(* IEC 61131-3 sources: generating_plc_code_with_llms/Code#2/ChatGPT_3.5/first run, 21 files *)

(* ---- 14.st ---- *)
// 8.02s
// 2
FUNCTION FC1001 : BOOL
VAR_INPUT
	MEW: REAL;
	SP: REAL;
	HYS: REAL;
END_VAR

VAR_IN_OUT
	OUT: BOOL;
END_VAR

VAR
	P_HYS: REAL;
END_VAR

(* FC1001 function implementation *)
IF MEW > (SP + P_HYS) THEN
    OUT := TRUE;
ELSIF MEW < (SP - P_HYS) THEN
    OUT := FALSE;
END_IF;

(* Update the hysteresis for the next cycle *)
P_HYS := SP * HYS / 100;

(* Return the output state *)
RETURN OUT;

(* ---- 15.st ---- *)
// 8.78s
// 2
FUNCTION FC1002 : BOOL
VAR_INPUT
	E_A, SENSOR: BOOL;
	ZEITW: TIME;
END_VAR

VAR_IN_OUT
	ZEIT: TON;
	P_HU, P_AL: BOOL;
END_VAR

(* FC1002 function implementation *)
IF E_A THEN
    IF SENSOR THEN
        ZEIT(IN := TRUE, PT := ZEITW);
        P_HU := NOT ZEIT.Q;
        P_AL := ZEIT.Q;
    ELSE
        ZEIT(IN := FALSE);
        P_HU := FALSE;
        P_AL := FALSE;
    END_IF;
ELSE
    ZEIT(IN := FALSE);
    P_HU := FALSE;
    P_AL := FALSE;
END_IF;

(* Return the output state *)
RETURN E_A;

(* ---- 18.st ---- *)
// 7.1s
// 4
FUNCTION FC1003 : VOID
VAR_INPUT
    IN_R: REAL;
    IN_MAX, IN_MIN: REAL;
    OUT_MAX, OUT_MIN: REAL;
END_VAR
VAR_OUTPUT
    OUT_R: REAL;
    FEH: BOOL;
END_VAR
VAR_TEMP
    DIFF1, DIFF2: REAL;
END_VAR

(* Check if input is within the specified range *)
IF (IN_R >= IN_MIN) AND (IN_R <= IN_MAX) THEN
    (* Calculate the differences between the input and output ranges *)
    DIFF1 := OUT_MAX - OUT_MIN;
    DIFF2 := IN_MAX - IN_MIN;

    (* Calculate the scaled temperature value within the output range *)
    OUT_R := OUT_MIN + ((IN_R - IN_MIN) / DIFF2) * DIFF1;

    (* Set FEH (Function Executed Healthy) to TRUE *)
    FEH := TRUE;
ELSE
    (* Set FEH to FALSE if input is outside the specified range *)
    FEH := FALSE;
END_IF

(* ---- 19.st ---- *)
// 10.82s
// 2
FUNCTION_BLOCK FB1005
VAR_INPUT
    START: BOOL;
    DICKE, V_MAX, V_MIN: REAL;
END_VAR

VAR_OUTPUT
    D_MAX, D_MIN: REAL;
    P1: BOOL;
END_VAR

VAR
    FO: BOOL;
    M_MAX, M_MIN: REAL;
END_VAR

METHOD CheckThickness: BOOL
VAR_INPUT
    S1: BOOL;
END_VAR
VAR
    CurrentThickness: REAL;
BEGIN
    (* Check if the sensor is active *)
    IF S1 THEN
        (* Calculate the thickness from the difference of laser measurements *)
        CurrentThickness := DICKE;

        (* Update the maximum and minimum thickness values *)
        IF CurrentThickness > M_MAX THEN
            M_MAX := CurrentThickness;
        END_IF;

        IF CurrentThickness < M_MIN THEN
            M_MIN := CurrentThickness;
        END_IF;

        (* Check if the current thickness is outside the tolerance band *)
        IF CurrentThickness > V_MAX OR CurrentThickness < V_MIN THEN
            P1 := TRUE; (* Switch on the reject light *)
        ELSE
            P1 := FALSE; (* Switch off the reject light *)
        END_IF;
    END_IF;

    (* Output the maximum and minimum thickness values *)
    D_MAX := M_MAX;
    D_MIN := M_MIN;

    (* Reset the thickness values at the start of a new measurement *)
    IF NOT S1 THEN
        M_MAX := 0.0;
        M_MIN := 9999.0; (* Assign an initial large value for comparison *)
    END_IF;

    (* Return the status of the reject light *)
    RETURN P1;
END_METHOD

END_FUNCTION_BLOCK

(* ---- 20.st ---- *)
// 11.08s
// 2
FUNCTION_BLOCK INTERLOCK
    VAR_INPUT
        I1: BOOL;
        I2: BOOL;
        TL: TIME;
    END_VAR

    VAR_OUTPUT
        Q1: BOOL;
        Q2: BOOL;
    END_VAR

    VAR
        T1: TOF(TL);
        T2: TOF(TL);
    END_VAR

    (* Interlock logic *)
    T1(IN:=NOT Q2 AND I1);
    T2(IN:=NOT Q1 AND I2);

    Q1 := T1.Q;
    Q2 := T2.Q;

END_FUNCTION_BLOCK

(* ---- 21.st ---- *)
// 47.97s
// weiter generieren
// 2
FUNCTION_BLOCK BURNER
VAR_INPUT
    IN: BOOL;
    STAGE2: BOOL;
    OVER_TEMP: BOOL;
    OIL_TEMP: BOOL := TRUE;
    FLAME: BOOL;
    RST: BOOL;
    RST_TIMER: BOOL;
    PRE_HEAT_TIME: TIME := t#5s;
    PRE_VENT_TIME: TIME := t#15s;
    PRE_IGNITE_TIME: TIME := t#15s;
    POST_IGNITE_TIME: TIME := t#25s;
    STAGE2_DELAY: TIME := t#10s;
    SAFETY_TIME: TIME := t#5s;
    LOCKOUT_TIME: TIME := t#10s;
    MULTIPLE_IGNITION: BOOL := TRUE;
    KW1: REAL;
    KW2: REAL;
END_VAR
VAR_OUTPUT
    MOTOR: BOOL;
    COIL1: BOOL;
    COIL2: BOOL;
    PRE_HEAT: BOOL;
    IGNITE: BOOL;
    FAIL: BOOL;
    KWH: REAL;
    STATUS: BYTE;
END_VAR
VAR_IN_OUT
    RUNTIME1: UDINT;
    RUNTIME2: UDINT;
    CYCLES: UDINT;
END_VAR
VAR
    state: INT;
    last: TIME;
    tx: TIME;
    last_change: TIME;
    timer1: TON;
    timer2: TON;
    oil_temp_last: BOOL;
    cycles2: UDINT;
END_VAR

METHOD BurnerControl: BOOL
    (* Internal Function to Control Burner *)
    VAR
        t1, t2, t3, t4, t5, t6: TIME;
    END_VAR

    t1 := PRE_HEAT_TIME;
    t2 := t1 + PRE_VENT_TIME;
    t3 := t2 + PRE_IGNITE_TIME;
    t4 := t3 + SAFETY_TIME;
    t5 := t4 + POST_IGNITE_TIME;
    t6 := t5 + STAGE2_DELAY;

    CASE state OF
        110:
            (* Wait for Start Signal (Standby) *)
            IF IN THEN
                state := 111;  (* Move to Startup Sequence *)
                last_change := tx;
            END_IF;
        111:
            (* Startup Sequence *)
            IF NOT OVER_TEMP THEN
                IF (NOT MULTIPLE_IGNITION AND timer1.IN) OR (MULTIPLE_IGNITION) THEN
                    (* Fuel Oil Warming *)
                    PRE_HEAT := TRUE;
                    IF (NOT OIL_TEMP AND (tx - last_change) <= PRE_HEAT_TIME) THEN
                        FAIL := TRUE;  (* Error: Fuel Oil Warming not responded within PRE_HEAT_TIME *)
                        STATUS := 1;
                        RETURN FALSE;
                    END_IF;
                    PRE_HEAT := FALSE;
                ELSE
                    FAIL := TRUE;  (* Error: Flame Sensor active during Fuel Oil Warming *)
                    STATUS := 2;
                    RETURN FALSE;
                END_IF;

                (* Pre-Purge (PRE_VENT_TIME) *)
                MOTOR := TRUE;
                COIL1 := TRUE;
                timer1(IN := TRUE, PT := t2);
                IF (FLAME AND (tx - last_change) <= PRE_VENT_TIME) THEN
                    FAIL := TRUE;  (* Error: Flame Sensor active during Pre-Purge *)
                    STATUS := 3;
                    RETURN FALSE;
                END_IF;

                (* Ignition *)
                COIL1 := FALSE;
                COIL2 := TRUE;
                IGNITE := TRUE;
                timer1(IN := TRUE, PT := t3);
                IF (NOT FLAME AND (tx - last_change) >= SAFETY_TIME) THEN
                    FAIL := TRUE;  (* Error: Safety time passed without flame *)
                    STATUS := 4;
                    RETURN FALSE;
                END_IF;
                IGNITE := FALSE;
                COIL2 := FALSE;
            END_IF;

            (* Stage 1 *)
            IF (tx - last_change) >= t4 THEN
                state := 112;
                last_change := tx;
            END_IF;
        112:
            (* Burner runs at Stage 1 *)
            MOTOR := TRUE;
            COIL1 := TRUE;
            timer1(IN := TRUE);
            KWH := KWH + KW1 * timer1.PT;
            RUNTIME1 := timer1.ET;
            IF (NOT FLAME) THEN
                FAIL := TRUE;  (* Error: Flame stops in operation *)
                STATUS := 5;
                RETURN FALSE;
            END_IF;

            (* Multiple Ignition *)
            IF (FLAME AND MULTIPLE_IGNITION AND (tx - last_change) <= POST_IGNITE_TIME) THEN
                state := 111;  (* Immediately start ignition for stage 1 *)
            END_IF;

            (* Stage 2 Activation *)
            IF STAGE2 AND (tx - last_change) >= t6 THEN
                state := 113;
                last_change := tx;
            END_IF;
        113:
            (* Burner runs at Stage 2 *)
            MOTOR := TRUE;
            COIL2 := TRUE;
            timer2(IN := TRUE);
            KWH := KWH + KW2 * timer2.PT;
            RUNTIME2 := timer2.ET;
    END_CASE;

    (* Check for RST (Reset) *)
    IF RST THEN
        IF (tx - last_change) >= LOCKOUT_TIME AND NOT RST_TIMER THEN
            RST_TIMER := TRUE;  (* Lockout Time Passed, Allow Reset *)
        END_IF;

        IF RST_TIMER THEN
            state := 110;  (* Reset, return to Standby *)
            last_change := tx;
            RST_TIMER := FALSE;
            CYCLES := CYCLES + 1;
        END_IF;
    END_IF;

    (* Check for Over-Temperature *)
    IF OVER_TEMP THEN
        state := 110;  (* Stop immediately every action and report error 9 *)
        FAIL := TRUE;
        STATUS := 9;
    END_IF;

    (* Update STATUS Output *)
    CASE state OF
        110: STATUS := 110;
        111: STATUS := 111;
        112: STATUS := 112;
        113: STATUS := 113;
    END_CASE;

    RETURN TRUE;
END_METHOD;

(* ---- 1.st ---- *)
// 6.53s
// 3
VAR
    xAllOn : BOOL;
    xAllOff : BOOL;

    xAlarm1 : BOOL;
    xAlarm2 : BOOL;
END_VAR

xAllOn := FALSE;
xAllOff := FALSE;
xAlarm1 := FALSE;
xAlarm2 := FALSE;

IF xAllOn THEN
    xAlarm1 := TRUE;
    xAlarm2 := TRUE;
    xAllOn := FALSE;  (* Turn off the xAllOn signal *)
END_IF;

IF xAllOff THEN
    xAlarm1 := FALSE;
    xAlarm2 := FALSE;
    xAllOff := FALSE;  (* Turn off the xAllOff signal *)
END_IF;

(* ---- 10.st ---- *)
// 5.01s
// 4
VAR_INPUT
    X : REAL;
END_VAR

VAR
    result : REAL;
END_VAR

(* Sigmoid function implementation *)
result := 1.0 / (1.0 + EXP(-X));

(* ---- 11.st ---- *)
// 4.88s
// 4
VAR_INPUT
    x : REAL;
END_VAR

VAR
    result : INT;
END_VAR

(* Sign function implementation *)
IF x > 0 THEN
    result := 1;
ELSIF x < 0 THEN
    result := -1;
ELSE
    result := 0;
END_IF;

(* ---- 12.st ---- *)
// 5.26s
// 4
VAR
    X : REAL;
END_VAR

VAR
    result : REAL;
END_VAR

(* Hyperbolic sine function implementation *)
result := (EXP(X) - EXP(-X)) / 2.0;

(* ---- 13.st ---- *)
// 7.85s
// 2
VAR CONSTANT
    MAXNUMBERS : UINT := 99;
END_VAR

VAR
    aNumbers : ARRAY[0..MAXNUMBERS] OF INT;
    nCnt : INT;
END_VAR

VAR
    NumberToFind : INT := 10;
    bNumberFound : BOOL := FALSE;
END_VAR

(* Initialize array with random numbers for illustration purposes *)
FOR nCnt := 0 TO MAXNUMBERS DO
    aNumbers[nCnt] := RAND(1, 20); (* Replace with actual logic for generating random numbers *)
END_FOR;

(* Search for the specific number in the list *)
nCnt := 0;
REPEAT
    IF aNumbers[nCnt] = NumberToFind THEN
        bNumberFound := TRUE;
        EXIT;
    END_IF;
    nCnt := nCnt + 1;
UNTIL nCnt > MAXNUMBERS OR bNumberFound;

(* Check if the number was found or the end of the list is reached *)
IF bNumberFound THEN
    (* Number found *)
    // Your logic here
ELSE
    (* Number not found in the list *)
    // Your logic here
END_IF;

(* ---- 16.st ---- *)
// 12.43s
// 2
VAR
    North_green : BOOL;
    North_yellow : BOOL;
    North_red : BOOL;
    East_green : BOOL;
    East_yellow : BOOL;
    East_red : BOOL;
    T1 : TON;
END_VAR

T1(IN:=TRUE, PT:=10000); (* 10-second cycle *)

IF T1.Q THEN
    (* Between 0ms and 5000ms *)
    IF T1.ET < 5000 THEN
        North_green := TRUE;
        North_yellow := FALSE;
        North_red := FALSE;
        East_green := FALSE;
        East_yellow := FALSE;
        East_red := TRUE;

    (* Between 5000ms and 5500ms *)
    ELSIF T1.ET < 5500 THEN
        North_green := FALSE;
        North_yellow := TRUE;
        North_red := FALSE;
        East_green := FALSE;
        East_yellow := FALSE;
        East_red := TRUE;

    (* Between 5500ms and 9500ms *)
    ELSIF T1.ET < 9500 THEN
        North_green := FALSE;
        North_yellow := FALSE;
        North_red := TRUE;
        East_green := TRUE;
        East_yellow := FALSE;
        East_red := FALSE;

    (* Between 9500ms and 10000ms *)
    ELSE
        North_green := FALSE;
        North_yellow := FALSE;
        North_red := TRUE;
        East_green := FALSE;
        East_yellow := TRUE;
        East_red := FALSE;
    END_IF;
ELSE
    (* Reset lights when the timer is not active *)
    North_green := FALSE;
    North_yellow := FALSE;
    North_red := FALSE;
    East_green := FALSE;
    East_yellow := FALSE;
    East_red := FALSE;
END_IF

(* ---- 17.st ---- *)
// 6.11s
// 4
VAR
    aiOutside : INT;
    aiHumidity: INT;
    sShowText : STRING[80];
END_VAR

(* Weather station program *)
IF aiOutside < 18 THEN
    sShowText := 'Cold';
ELSIF aiOutside >= 18 AND aiOutside <= 25 THEN
    IF aiHumidity >= 40 AND aiHumidity <= 75 THEN
        sShowText := 'Opt';
    ELSE
        sShowText := 'Temp. OK';
    END_IF;
ELSE
    sShowText := 'Hot';
END_IF;

(* ---- 2.st ---- *)
// 4.98s
// 4
VAR_INPUT
    N : INT;
    K : INT;
    i : INT;
END_VAR

VAR
    result : INT;
END_VAR

result := 1;

FOR i := 1 TO K DO
    result := result * (N - i + 1) / i;
END_FOR;

(* ---- 3.st ---- *)
// 5.44s
// 2
VAR_INPUT
    X : INT;
END_VAR

VAR
    t1 : DINT;
    t2 : DINT;
    x_tmp : INT;
END_VAR

t1 := 0;
t2 := 1;

IF X = 0 THEN
    x_tmp := t1;
ELSIF X = 1 THEN
    x_tmp := t2;
ELSE
    FOR i := 2 TO X DO
        x_tmp := t1 + t2;
        t1 := t2;
        t2 := x_tmp;
    END_FOR;
END_IF;

(* ---- 4.st ---- *)
// 8.35s
// 2
VAR
    aiLevel : INT;
    PercentLevel : UINT;
    doLow : BOOL;
    doOk : BOOL;
    doHigh : BOOL;
    doAlarm : BOOL;
END_VAR

CASE aiLevel OF
    (aiLevel <= 327) :
        PercentLevel := 0;
        doLow := TRUE;
        doOk := FALSE;
        doHigh := FALSE;
    (aiLevel > 327 AND aiLevel <= 1638) :
        PercentLevel := (aiLevel - 327) * 100 / (1638 - 327);
        doLow := FALSE;
        doOk := TRUE;
        doHigh := FALSE;
    (aiLevel > 1638 AND aiLevel <= 3111) :
        PercentLevel := (aiLevel - 1638) * 100 / (3111 - 1638);
        doLow := FALSE;
        doOk := TRUE;
        doHigh := FALSE;
    (aiLevel > 3111 AND aiLevel <= 32767) :
        PercentLevel := (aiLevel - 3111) * 100 / (32767 - 3111);
        doLow := FALSE;
        doOk := FALSE;
        doHigh := TRUE;
    TRUE :
        PercentLevel := 100;
        doLow := FALSE;
        doOk := FALSE;
        doHigh := TRUE;
END_CASE;

IF PercentLevel < 1 THEN
    doAlarm := TRUE;
ELSE
    doAlarm := FALSE;
END_IF;

(* ---- 5.st ---- *)
// 6.9s
// 3
VAR
    Start_Loop : BOOL := FALSE;
    one_hour : TIME := T#1h;
    One_Hour_Timer : TON;
    Gate_Open : BOOL := FALSE;
    Close_Gate_Inst : BOOL := FALSE;
    Sensed_Car : BOOL := FALSE;
    Sensed_Car_Inst : BOOL := FALSE;
    Sensed_App : BOOL := FALSE;
    Mobile_Inst : BOOL := FALSE;
    Auth : STRING;
    my_defined_str : STRING := 'abcd';
END_VAR

One_Hour_Timer(IN := NOT Start_Loop, PT := one_hour);
Close_Gate_Inst := One_Hour_Timer.Q;

IF Close_Gate_Inst THEN
    IF Gate_Open THEN
        Gate_Open := FALSE;
    END_IF;
END_IF;

IF Sensed_Car AND Sensed_Car_Inst AND Auth = my_defined_str THEN
    Gate_Open := TRUE;
END_IF;

IF Sensed_App AND Mobile_Inst AND Auth = my_defined_str THEN
    Gate_Open := TRUE;
END_IF;

(* ---- 6.st ---- *)
// 11.59s
// 4
VAR CONSTANT
    WAIT : UINT := 0;
    TOP_POSITION : UINT := 1;
    BOTTOM_POSITION : UINT := 2;
    GETBOX : UINT := 3;
    UNLOAD_POSITION : UINT := 4;
    UNLOAD_BOX : UINT := 5;
END_VAR

VAR
    (*-- digital outputs*)
    doConvTop : BOOL;
    doConvBottom : BOOL;
    doConvLift : BOOL;
    doLiftTop : BOOL;
    doLiftBottom : BOOL;
    doLiftUnload : BOOL;
    (*-- digital inputs*)
    diConvTop : BOOL;
    diConvBottom : BOOL;
    diLiftTop : BOOL;
    diLiftBottom : BOOL;
    diLiftUnload : BOOL;
    diBoxLift : BOOL;
    (*-- status variables*)
    selectLift : UINT;
    ConvTopOn : BOOL;
    ConvBottomOn : BOOL;
END_VAR

CASE selectLift OF
    WAIT :
        ConvTopOn := FALSE;
        ConvBottomOn := FALSE;
        IF diConvTop THEN
            selectLift := TOP_POSITION;
        ELSIF diConvBottom THEN
            selectLift := BOTTOM_POSITION;
        END_IF;
    TOP_POSITION :
        doLiftTop := TRUE;
        doLiftBottom := FALSE;
        IF diLiftTop THEN
            selectLift := GETBOX;
        END_IF;
    BOTTOM_POSITION :
        doLiftTop := FALSE;
        doLiftBottom := TRUE;
        IF diLiftBottom THEN
            selectLift := GETBOX;
        END_IF;
    GETBOX :
        doConvLift := TRUE;
        IF diBoxLift THEN
            doConvLift := FALSE;
            selectLift := UNLOAD_POSITION;
        END_IF;
    UNLOAD_POSITION :
        doLiftUnload := TRUE;
        IF diLiftUnload THEN
            selectLift := UNLOAD_BOX;
        END_IF;
    UNLOAD_BOX :
        doLiftUnload := FALSE;
        selectLift := WAIT;
END_CASE;

(* Stop conveyor belts if requested by light barrier *)
doConvTop := NOT diConvTop AND NOT ConvTopOn;
doConvBottom := NOT diConvBottom AND NOT ConvBottomOn;

(* ---- 7.st ---- *)
// 6.29s
// 2
VAR CONSTANT
    MAX_INDEX : USINT := 4;
END_VAR

VAR
    aWeights : ARRAY[0..MAX_INDEX] OF INT;
    iCnt : USINT;
    sumWeight : DINT;
    avgWeight : INT;
END_VAR

sumWeight := 0;

FOR iCnt := 0 TO MAX_INDEX DO
    sumWeight := sumWeight + aWeights[iCnt];
END_FOR;

avgWeight := sumWeight / (MAX_INDEX + 1);

(* ---- 8.st ---- *)
// 7.38s
// 2
VAR_INPUT
    X : REAL;
END_VAR

VAR
    w : REAL;
    i : INT;
    we : REAL;
    w1e : REAL;
    ewx : REAL;
    last : DWORD;
END_VAR

CONSTANT
    MAX_ITERATIONS : INT := 50;
    EPSILON : REAL := 1.0E-8;
END_CONSTANT

w := X;

FOR i := 1 TO MAX_ITERATIONS DO
    ewx := EXP(w);
    we := w * ewx;
    w1e := w + 1.0;
    w := w - (we - X) / (w1e * ewx - (w + 2.0) * we / (2.0 * w1e));
    IF ABS(w - last) < EPSILON THEN
        EXIT;
    END_IF;
    last := w;
END_FOR;

(* ---- 9.st ---- *)
// 5.58s
// 3
VAR
    YEAR : INT;
END_VAR

VAR
    isLeapYear : BOOL := FALSE;
END_VAR

(* Check if the year is a leap year *)
IF YEAR MOD 4 = 0 THEN
    IF YEAR MOD 100 = 0 THEN
        IF YEAR MOD 400 = 0 THEN
            isLeapYear := TRUE;
        END_IF;
    ELSE
        isLeapYear := TRUE;
    END_IF;
END_IF;
